{attribute 'linkalways'} 
{attribute 'no_explicit_call' := 'This FB is a CLASS and must be accessed using methods or properties'}
{attribute 'enable_dynamic_creation'}
FUNCTION_BLOCK ContentAddedEvent EXTENDS Disposable IMPLEMENTS I_ContentAddedEvent
VAR
	_targetContent : I_Content;
END_VAR

METHOD FB_init : BOOL
VAR_INPUT
	bInitRetains : BOOL; // if TRUE, the retain variables are initialized (warm start / cold start)
	bInCopyCode : BOOL;  // if TRUE, the instance afterwards gets moved into the copy code (online change)
	TargetContent : I_Content;
END_VAR
This^._targetContent := TargetContent;
END_METHOD

PROPERTY PUBLIC TargetContent : I_Content
GET
TargetContent := _targetContent;
END_GET
END_PROPERTY

END_FUNCTION_BLOCK

(* stored: Version 1.1.0.1, ProductVersion 3.1.4024.12
   POU ContentAddedEvent: Id {f9599a83-968a-0135-07a6-7d7daeece167}, SpecialFunc None
   Folder Constructor: Id {08324144-5a6a-0c6a-0753-5673627f1b1a}
   Method FB_init: Id {9beb3ab6-e32f-0cb9-0ab4-210479bb5e0a}
   Property TargetContent: Id {3a25a44e-a50b-0719-38fb-df36651953ab}
   Get Get: Id {f522199a-d6de-0e4c-21c2-6dd6f80d69f7} *)
